(* Logix 5000 project; controller Ex_2_11 Emulate 5570 rev 33.11; software revision 33.00 *)
// Pacakge on conveyor belt

TASK MainTask (continuous, watchdog 500 ms) : MainProgram

MODULES
   Local : Emulate 5570 (ICP 4, rev 33.11)
END_MODULES

VAR_GLOBAL   (* controller tags *)
   B1 : BOOL;   // Sensor B1
   M1 : BOOL;   // Motor M1
   ONS_1 : BOOL;
   Pacakge_Online : BOOL;
   S1 : BOOL;   // Rotory Switch S1
   Start_Trigger : BOOL;
END_VAR

PROGRAM MainProgram   (* main routine MainRoutine *)

ROUTINE MainRoutine   (* ladder *)
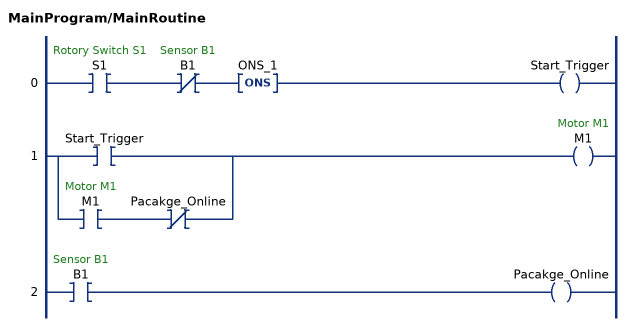
   0: XIC(S1)XIO(B1)ONS(ONS_1)OTE(Start_Trigger);
   1: [XIC(Start_Trigger) ,XIC(M1) XIO(Pacakge_Online) ]OTE(M1);
   2: XIC(B1)OTE(Pacakge_Online);
END_ROUTINE
END_PROGRAM
